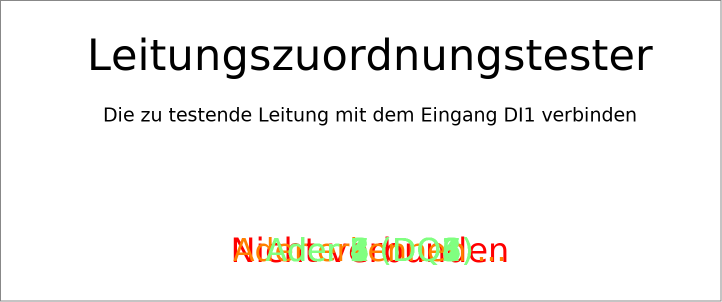
VISUALIZATION LeitungszuordnungsTester  // 722x302
    Label (20,20 700x70), "Leitungszuordnungstester"
    Label (20,100 700x30), "Die zu testende Leitung mit dem Eingang DI1 verbinden"
    Label (20,200 700x100), "Nicht verbunden", invisible if: NOT Visu.NichtVerbunden
    Label (20,200 700x100), "Ader erkennen ...", invisible if: NOT Visu.AderErkennen
    Label (20,200 700x100), "Ader 1 (DQ1)", invisible if: NOT Visu.Ader_1
    Label (20,200 700x100), "Ader 2 (DQ2)", invisible if: NOT Visu.Ader_2
    Label (20,200 700x100), "Ader 3 (DQ3)", invisible if: NOT Visu.Ader_3
    Label (20,200 700x100), "Ader 4 (DQ4)", invisible if: NOT Visu.Ader_4
    Label (20,200 700x100), "Ader 5 (DQ5)", invisible if: NOT Visu.Ader_5
    Label (20,200 700x100), "Ader 6 (DQ6)", invisible if: NOT Visu.Ader_6
    Label (20,200 700x100), "Ader 7 (DQ7)", invisible if: NOT Visu.Ader_7
    Label (20,200 700x100), "Ader 8 (DQ8)", invisible if: NOT Visu.Ader_8
END_VISUALIZATION

(* stored: Version 1.1.0.1, ProductVersion 3.1.4022.7
   Visu LeitungszuordnungsTester: Id {305e9e29-6495-4dae-bfb3-a6962cf59250} *)
